FUNCTION_BLOCK Override_K_Select (* Aktiv/Wert (AX) zu K (AUI) fuer AX_AUI_MUX_3: 0=Normal, 1=Force FALSE, 2=Force TRUE *)
  (* Standard: 61499-2; Description: Copyright (c) 2026 HR Agrartechnik GmbH This program and the accompanying materials are made available under the terms of the Eclipse Public License 2.0 which is available at https://www.eclipse.org/legal/epl-2.0/ SPDX-License-Identifier: EPL-2.0 *)
  (* Version 1.0, 2026-08-13, Franz Höpfinger, HR Agrartechnik GmbH, initial API and implementation *)
  PACKAGE adapter::OverrideK;
  IMPORT adapter::OverrideK::const::Override_K::Override_K_Normal;
  IMPORT adapter::OverrideK::const::Override_K::Override_K_ForceFalse;
  IMPORT adapter::OverrideK::const::Override_K::Override_K_ForceTrue;
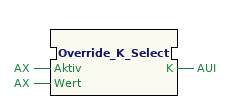
  SOCKETS
    Aktiv : adapter::types::unidirectional::AX; (* Override.Aktiv *)
    Wert : adapter::types::unidirectional::AX; (* Override.Wert *)
  END_SOCKETS
  PLUGS
    K : adapter::types::unidirectional::AUI; (* 0=Normal (Aktiv=FALSE), 1=Force FALSE (Aktiv=TRUE, Wert=FALSE), 2=Force TRUE (Aktiv=TRUE, Wert=TRUE) *)
  END_PLUGS
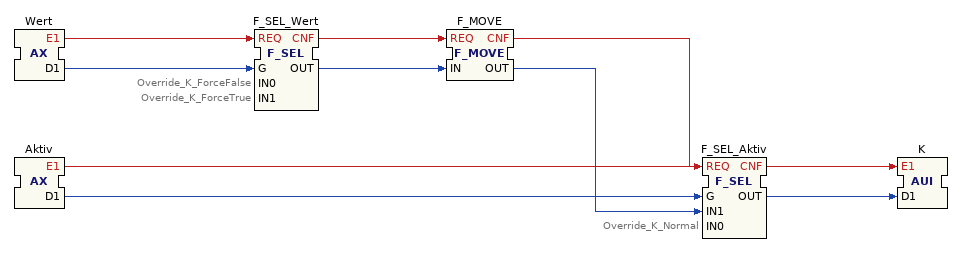
  FBS
    F_SEL_Wert : iec61131::selection::F_SEL(IN0 := Override_K_ForceFalse, IN1 := Override_K_ForceTrue);
    F_SEL_Aktiv : iec61131::selection::F_SEL(IN0 := Override_K_Normal);
    F_MOVE : iec61131::selection::F_MOVE; {SET_ATTRIBUTE(DataType, UINT)}
  END_FBS
  EVENT_CONNECTIONS
    Wert.E1 TO F_SEL_Wert.REQ;
    Aktiv.E1 TO F_SEL_Aktiv.REQ;
    F_SEL_Aktiv.CNF TO K.E1;
    F_SEL_Wert.CNF TO F_MOVE.REQ;
    F_MOVE.CNF TO F_SEL_Aktiv.REQ;
  END_CONNECTIONS
  DATA_CONNECTIONS
    Wert.D1 TO F_SEL_Wert.G;
    Aktiv.D1 TO F_SEL_Aktiv.G;
    F_SEL_Wert.OUT TO F_MOVE.IN;
    F_SEL_Aktiv.OUT TO K.D1;
    F_MOVE.OUT TO F_SEL_Aktiv.IN1;
  END_CONNECTIONS
END_FUNCTION_BLOCK
